Staubli VAL3: clear.pgx

public program clear()
begin
  nElems = 0
  nPush = nPop
end
